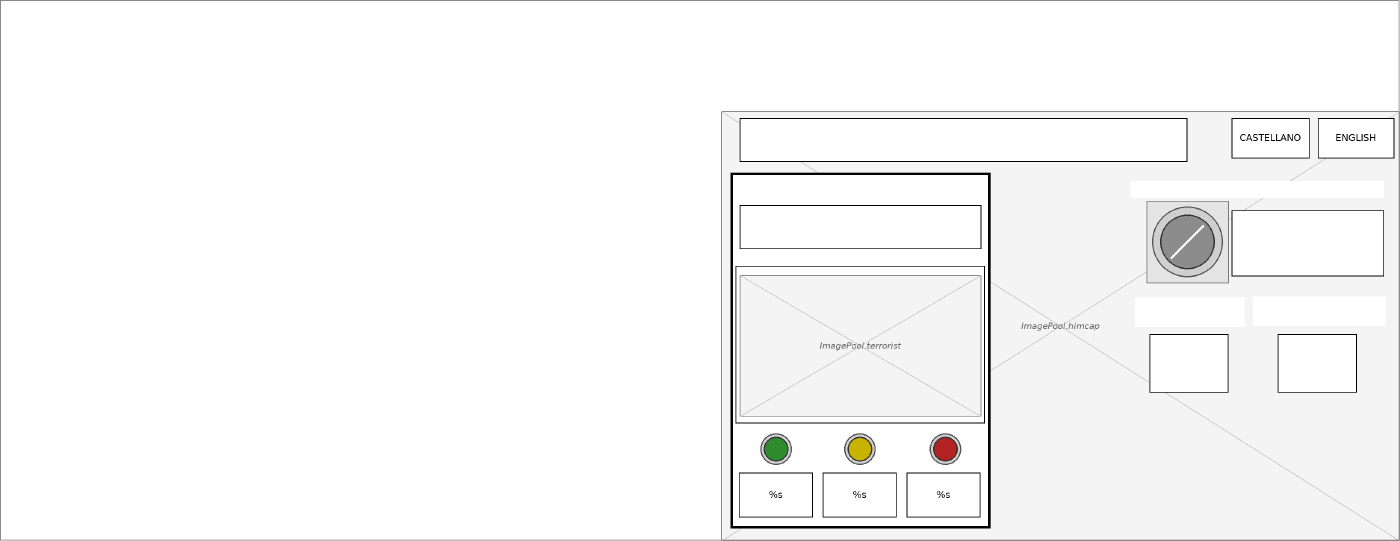
VISUALIZATION HMI  // 1637x633
    Image (843,130 794x503), image: ImagePool.himcap
    RoundedRectangle (854,202 304x416)
    Rectangle (860,311 291x184)
    Image (865,322 282x165), image: ImagePool.terrorist
        p84334746: MAIN.HMI_CTRL.sImagenActual
    RotarySwitch (1339,235 99x96), variable: MAIN.EMERGENCY_HDL.stSystem.inputs.iSwitch_HMI, behaviour: TOGGLE, style: Switch-RotarySwitch-Gray
    RoundedRectangle (1494,391 92x68)
        tap MAIN.EMERGENCY_HDL.stSystem.inputs.iTestButton_HMI
    RoundedRectangle (1344,391 92x68)
        toggle MAIN.EMERGENCY_HDL.stSystem.inputs.iAlarmButton_HMI
    Rectangle (1327,348 128x34), "%s", text list: 'TextList', text index: 6
    Rectangle (1322,212 296x19), "%s", text list: 'TextList', text index: 5
    Lamp1 (886,503 43x45), variable: MAIN.stSystem.outputs.oLightGreen, style: Lamp-Lamp1-Green
    Lamp1 (984,503 43x45), variable: MAIN.stSystem.outputs.oLightOrange, style: Lamp-Lamp1-Yellow
    Lamp1 (1084,503 43x45), variable: MAIN.stSystem.outputs.oLightRed, style: Lamp-Lamp1-Red
    RoundedRectangle (864,553 86x52), "%s", text list: 'TextList', text index: 2
    RoundedRectangle (962,553 86x52), "%s", text list: 'TextList', text index: 3
    RoundedRectangle (1060,553 86x52), "%s", text list: 'TextList', text index: 4
    Rectangle (1465,347 155x34), "%s", text list: 'TextList', text index: 7
    Rectangle (865,240 282x51), "%s", text list: 'TextList', text index: 1
    RoundedRectangle (1541,138 89x47), "ENGLISH"
        OnMouseClick: ChangeLanguage ChangeLanguage=English
    RoundedRectangle (1440,138 91x47), "CASTELLANO"
        OnMouseClick: ChangeLanguage ChangeLanguage=Spanish
    Rectangle (1440,246 178x77), "%s", text list: 'TextList', text index: 0
    Rectangle (865,138 523x51), "%s", text list: 'TextList', text index: 9
END_VISUALIZATION

(* stored: Version 1.1.0.1, ProductVersion 3.1.4026.12
   Visu HMI: Id {3ab4dd97-cc29-4641-81f9-abe1c84ad934} *)
